(* IEC 61131-3 sources: repolevel_ST_code_completion/dataset/project_code/SRCI-main/FUN, 1 file *)

(* ---- CheckBounds.st ---- *)
// Implicitly generated code : DO NOT EDIT
FUNCTION CheckBounds : DINT
VAR_INPUT
  index, lower, upper: DINT;
END_VAR

// Implicitly generated code : Only an Implementation suggestion
{noflow}
IF  index < lower THEN
  CheckBounds := lower;
ELSIF  index > upper THEN
  CheckBounds := upper;
ELSE
  CheckBounds := index;
END_IF
{flow}
